// TIA Portal V19 export
FUNCTION_BLOCK "Check_Axis_Velocity"   // FB189, LAD
TITLE = CHECK AXIS VELOCITY USING POSITION VARIATION
// stored: Access Published, MemoryReserve 100, SetENOAutomatically false
   VAR_INPUT
      AcualPosition : LReal;
      PositionModule : LReal;
      StandstillVelocityThreshold : LReal := 200.0;
   END_VAR
   VAR_OUTPUT
      LessThanStandstillThreshold : Bool;
      VelocityCalculated : LReal;
   END_VAR
   VAR
      Sts : Struct
         Act_Time : DTL;
         Prv_Time : DTL;
         Act_Pos : LReal;
         Prv_Pos : LReal;
         Delta_Time : Time;
         Delta_T : LReal;
         Delta_S : LReal;
      END_STRUCT;
   END_VAR
   VAR_TEMP
      ReturnValue : Word;
   END_VAR
   VAR_TEMP   // added for the SCL form of the ladder/FBD networks
      _w1 : Bool;
   END_VAR
BEGIN

REGION Network 1: Delta Time in minutes
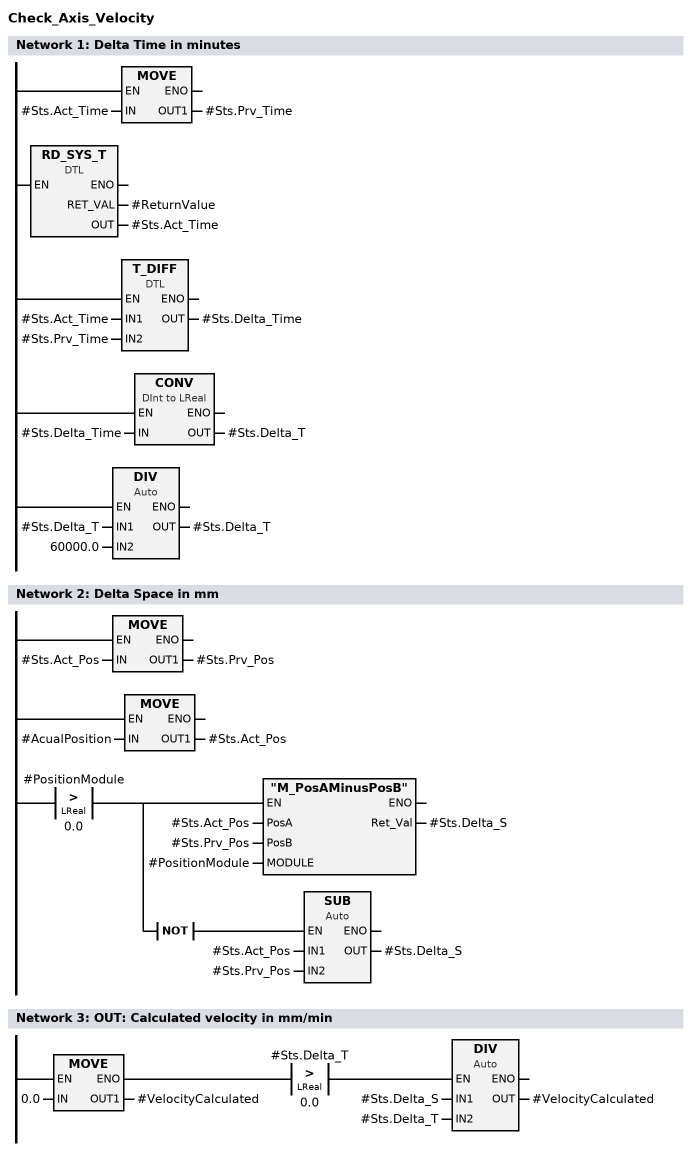
   RUNG wire#powerrail
      { S7_GenerateENO := "TRUE" } Move(in := #Sts.Act_Time, out1 => #Sts.Prv_Time)
   END_RUNG
   RUNG wire#powerrail
      { S7_Templates := "date_type := DTL" } RD_SYS_T(RET_VAL => #ReturnValue, OUT => #Sts.Act_Time)
   END_RUNG
   RUNG wire#powerrail
      { S7_Templates := "[date_type := DTL, time_type := Time]" } T_DIFF(IN1 := #Sts.Act_Time, IN2 := #Sts.Prv_Time, OUT => #Sts.Delta_Time)
   END_RUNG
   RUNG wire#powerrail
      { S7_Templates := "[SrcType := DInt, DestType := LReal]"; S7_GenerateENO := "TRUE" } Convert(in := #Sts.Delta_Time, out => #Sts.Delta_T)
   END_RUNG
   RUNG wire#powerrail
      { S7_GenerateENO := "TRUE" } Div(in1 := #Sts.Delta_T, in2 := 60000.0, out => #Sts.Delta_T)
   END_RUNG
   // the same network as SCL:
   #Sts.Prv_Time := #Sts.Act_Time;
   #ReturnValue := RD_SYS_T(OUT => #Sts.Act_Time);
   T_DIFF(IN1 := #Sts.Act_Time, IN2 := #Sts.Prv_Time, OUT => #Sts.Delta_Time);
   #Sts.Delta_T := DINT_TO_LREAL(#Sts.Delta_Time);
   #Sts.Delta_T := #Sts.Delta_T / 60000.0;
END_REGION

REGION Network 2: Delta Space in mm
   RUNG wire#powerrail
      { S7_GenerateENO := "TRUE" } Move(in := #Sts.Act_Pos, out1 => #Sts.Prv_Pos)
   END_RUNG
   RUNG wire#powerrail
      { S7_GenerateENO := "TRUE" } Move(in := #AcualPosition, out1 => #Sts.Act_Pos)
   END_RUNG
   RUNG wire#powerrail
      { S7_Templates := "SrcType := LReal" } GT_Contact(in1 := #PositionModule, in2 := 0.0)
      wire#w1
      "M_PosAMinusPosB"(PosA := #Sts.Act_Pos, PosB := #Sts.Prv_Pos, MODULE := #PositionModule, Ret_Val => #Sts.Delta_S)
   END_RUNG
   RUNG wire#w1
      Not()
      { S7_GenerateENO := "TRUE" } Sub(in1 := #Sts.Act_Pos, in2 := #Sts.Prv_Pos, out => #Sts.Delta_S)
   END_RUNG
   // the same network as SCL:
   #Sts.Prv_Pos := #Sts.Act_Pos;
   #Sts.Act_Pos := #AcualPosition;
   #_w1 := #PositionModule > 0.0;
   IF #_w1 THEN
       #Sts.Delta_S := "M_PosAMinusPosB"(PosA := #Sts.Act_Pos, PosB := #Sts.Prv_Pos, MODULE := #PositionModule);
   END_IF;
   IF NOT #_w1 THEN #Sts.Delta_S := #Sts.Act_Pos - #Sts.Prv_Pos; END_IF;
END_REGION

REGION Network 3: OUT: Calculated velocity in mm/min
   RUNG wire#powerrail
      { S7_GenerateENO := "TRUE" } Move(in := 0.0, out1 => #VelocityCalculated)
      { S7_Templates := "SrcType := LReal" } GT_Contact(in1 := #Sts.Delta_T, in2 := 0.0)
      { S7_GenerateENO := "TRUE" } Div(in1 := #Sts.Delta_S, in2 := #Sts.Delta_T, out => #VelocityCalculated)
   END_RUNG
   // the same network as SCL:
   // ENO of a box is taken as its EN; it also drops when the box reports an error
   #VelocityCalculated := 0.0;
   IF #Sts.Delta_T > 0.0 THEN #VelocityCalculated := #Sts.Delta_S / #Sts.Delta_T; END_IF;
END_REGION

REGION Network 4 (SCL): OUT: Velocity less then standstill threshold
   #LessThanStandstillThreshold := ABS(#VelocityCalculated) <= #StandstillVelocityThreshold;
END_REGION

REGION Network 5: +
END_REGION

REGION Network 6: +
END_REGION

REGION Network 7: +
END_REGION
END_FUNCTION_BLOCK
